FUNCTION_BLOCK FB_Logger
VAR_INPUT
	eLogLevel		: E_LogLevel;
	sMessage		: T_MaxString;
	stArg1			: T_Arg;
	stArg2			: T_Arg;
	stArg3			: T_Arg;	
	iContextBuilder	: I_ContextBuilder;	
END_VAR

METHOD FB_init : BOOL
VAR_INPUT
	bInitRetains : BOOL; // if TRUE, the retain variables are initialized (warm start / cold start)
	bInCopyCode : BOOL;  // if TRUE, the instance afterwards gets moved into the copy code (online change)
	sLogger		: T_MaxString;
END_VAR
END_METHOD

END_FUNCTION_BLOCK

(* stored: Version 1.1.0.1, ProductVersion 3.1.4024.0
   POU FB_Logger: Id {50b11db4-e622-4fbf-aac9-873d9c447954}, SpecialFunc None
   Method FB_init: Id {4f993583-02a7-4efe-804b-13cea4cdd5af} *)
